(* CoDeSys 2.3.8.0 project: Laser_G67HP_2.pro *)
(* Libraries: STANDARD.LIB 5.6.98 12:03:02 *)

(* Global variable list: Globale_Variablen *)
VAR_GLOBAL

	(* Hardwareeingänge *)
	INot_Aus 			 	AT %IX0.0 : BOOL; (* Eingang 1 *)
	IDruckW			  	AT %IX0.1 : BOOL; (* Eingang 2 *)
	ISchututuer	  		AT %IX0.2 : BOOL; (* Eingang 3 *)
	ISchutzhaube  		AT %IX0.3 : BOOL; (* Eingang 4 *)
	IHWT_EIN			 	AT %IX0.4 : BOOL; (* Eingang 5 *)
	IHWT_AUS			AT %IX0.5 : BOOL; (* Eingang 6 *)
	IHWT_Quitt  			AT %IX0.6 : BOOL; (* Eingang 7 *)
	IRES1					AT %IX0.7 : BOOL; (* Eingang 8 *)

       IINI_Ueberlast  		AT %IX1.0 : BOOL; (* Eingang 9 *)
	IINI_IndexVor	  		AT %IX1.1 : BOOL; (* Eingang 10 *)
	IINI_IndexRueck  		AT %IX1.2 : BOOL; (* Eingang 11 *)
	IINI_Kupplung  		AT %IX1.3 : BOOL; (* Eingang 12 *)
	IRES2			  		AT %IX1.4 : BOOL; (* Eingang 13 *)
	IRES3		 			AT %IX1.5 : BOOL; (* Eingang 14 *)
	IRES4					AT %IX1.6 : BOOL;
	IRES5		 			AT %IX1.7 : BOOL;

	IKammError  			AT %IX2.0 : BOOL; (* Eingang 17 *)
	IKammEnable  		AT %IX2.1 : BOOL; (* Eingang 18 *)
	IKammOutput  		AT %IX2.2 : BOOL; (* Eingang 19 *)
	IRES6		 			AT %IX2.3 : BOOL; (* Eingang 20 *)
	IAbsaug100P 			AT %IX2.4 : BOOL; (* Eingang 21 *)
	IAbsaugFilter			AT %IX2.5 : BOOL; (* Eingang 22 *)
	IRES					AT %IX2.6 : BOOL; (* Eingang 23 *)
	IFU_BB				AT %IX2.7 : BOOL; (* Eingang 24 *)

	IFrgMoma1 			AT %IX3.0 : BOOL;
	IFrgMoma2 			AT %IX3.1 : BOOL;
	IRES7	 				AT %IX3.2 : BOOL;
	IRES8	 				AT %IX3.3 : BOOL;
	ILAS_HWIO 			AT %IX3.4 : BOOL;
	ILAS_SWIO 			AT %IX3.5 : BOOL;
	ILAS_Redy	 		AT %IX3.6 : BOOL;
	ILAS_Res	 			AT %IX3.7 : BOOL;

	ILasDataBit0 			AT %IX4.0 : BOOL;
	ILasDataBit1 	 		AT %IX4.1 : BOOL;
	ILasDataBit2 		 	AT %IX4.2 : BOOL;
	ILasDataBit3 		 	AT %IX4.3 : BOOL;
	ILasDataBit4 	 		AT %IX4.4 : BOOL;
	ILasDataBit5 	 		AT %IX4.5 : BOOL;
	ILasResI1	 		 	AT %IX4.6 : BOOL;
	ILasResI2 			 	AT %IX4.7 : BOOL;

	(*Eingänge für die Panel Tasten*)

	IAPosKS1Input  		AT%IW20:INT;	 	(*Speicher 1 Füllstand analoger Eingang*)
	IARES1				AT%IW22:INT;
	IASSIDgInput			 AT %ID44:UDINT;	(* Drehgeber *)


	QHAmpelGn		 	AT %QX0.0 : BOOL; (* Ventil Pneumatik  *)
	QHAmpelRt	  		AT %QX0.1 : BOOL; (* Ausgang 2 *)
	QHAmpelGb 			AT %QX0.2 : BOOL; (* Ausgang 3 *)
	QRES1				AT %QX0.3 : BOOL; (* Ausgang 4 *)
	QHTasteEin			AT %QX0.4 : BOOL; (* Ausgang 5 *)
	QHTasteAus			AT %QX0.5 : BOOL; (* Ausgang 6 *)
	QHTasteQuitt			AT %QX0.6 : BOOL; (* Ausgang 7 *)
	QRES2				AT %QX0.7 : BOOL; (* Ausgang 8 *)

	QLasMark				AT %QX1.0 : BOOL; (* Ausgang 9 *)
	QLasMarkstop		AT %QX1.1 : BOOL; (* Ausgang 10 *)
	QLasProg1			AT %QX1.2 : BOOL; (* Ausgang 11 *)
	QLasProg2			AT %QX1.3 : BOOL; (* Ausgang 12 *)
	QLasRes2			AT %QX1.4 : BOOL; (* Ausgang 13 *)
	QLasRes3			AT %QX1.5 : BOOL; (* Ausgang 14 *)
	QFrgNaechst			AT %QX1.6 : BOOL; (* Ausgang 15 *)
	QAntriebeEin		     	AT %QX1.7 : BOOL; (* Ausgang 16 *)

	QMotVor	 			AT %QX2.0 : BOOL; (* Ausgang 9 *)
	QMotRueck			AT %QX2.1 : BOOL; (* Ausgang 10 *)
	QSaugAnford			AT %QX2.2 : BOOL; (* Ausgang 11 *)
	QVIndex				AT %QX2.3 : BOOL; (* Ausgang 12 *)
	QVUeberlast			AT %QX2.4 : BOOL; (* Ausgang 13 *)
	QRES5				AT %QX2.5 : BOOL; (* Ausgang 14 *)
	QRES6				AT %QX2.6 : BOOL; (* Ausgang 15 *)
	QRES7			     	AT %QX2.7 : BOOL; (* Ausgang 16 *)

	QASollwMot			AT%QW4:WORD; (*Ausgangswort 1*)
	QARes				 	AT%QW6:WORD; (*Ausgangswort 2*)

(* Anfang der Variablen für Kopmunikation SPS <> Visu *)
	TP_LaserAktiv	:		BOOL;
	TP_LaserHand:			BOOL;
	TP_RefSetzen:			BOOL;
	TP_KammeraAktiv:		BOOL;
	TP_MVor:				BOOL;
	TP_MVorS:				BOOL;
	TP_Mrueck:				BOOL;
	TP_MrueckS:				BOOL;
	TP_Hand:				BOOL;
	TP_Auto:					BOOL;
	TP_ZNullen:				BOOL;   (*not included yet*)
	TPTypIndex:				WORD; (*not included yet*)
	TPTypSpeichern:			BOOL;   (*not included yet*)
	TPKettenTyp: 			ARRAY[0..3] OF WORD;  (*not included yet*)

	S_StUeberlast:			BOOL;
	S_StLaser:				BOOL;
	S_StKammera:			BOOL;
	S_StKupplung	:			BOOL;
	S_StSpeicherSchutz:		BOOL;
	S_StLaserSchutz:			BOOL;
	S_StSpeicher:				BOOL;
	S_StSammelstoerung:	BOOL;
	S_StDruck:				BOOL;
	S_StNotAus:				BOOL;
	S_StRef:					BOOL;

	S_StSchutzTuer:  BOOL;
	S_StSchutzHaube : BOOL;
         S_StAbsaugFilter : BOOL;
         S_StAbsaug100p : BOOL;


	S_MSpeicherVoll:			BOOL;
	S_MSpeicherLeer:		BOOL;
	S_MWarteSpeicher:		BOOL;
	S_MHand:					BOOL;
	S_FKamera:				BOOL;
	S_FLaser:					BOOL;
	S_MAutoStart:				BOOL;
	S_MAutoStop:				BOOL;
	SI_Gliederzahl:			INT;
	SI_ProgNr:				INT;
	SI_IO:						INT;
	SI_NIO:					INT;
	SI_FPosLaser:			INT;
	SI_FPosKamera:			INT;
	SKettenTyp:ARRAY[0..3] OF WORD;  (*not included yet*)
(* ENDE*)

	Skal_IC_SSI_DG_Input: 	DINT;
	Skal_SSI_DG_4:			DINT;
	ZeigerReg:				INT;
	ZeigerKette: 				INT;
	ImpulsPos: 				BOOL;
	ImpulsNeg: 				BOOL;
	Sammelstoerung: BOOL;

	V_Erster_Zyklus: BOOL;
	REF_IO: BOOL;
	AktTypIndexAlt: WORD;
	AktTypindex:WORD;
	PosErreicht: BOOL;


END_VAR

VAR_GLOBAL RETAIN

	(* KettenTyp[0] = Gliederzahl,  Kettentyp[1] Farbe1 0=grau 1=gelb 2=rot 3=blau, Kettentyp[2]=position der ersten Farblasche (Nr.d. Außenlasche*)
	(*Kettentyp[3] Farbe2  Kettentyp[4] Position der zweiten Farblasche *)
	(*Kettentyp[6] Farbe3  Kettentyp[6] Position der dritten Farblasche *)
	(*Kettentyp[7] Farbe4  Kettentyp[8] Position der vierten Farblasche *)
	(*Kettentyp[9] Farbe5  Kettentyp[10] Position der fünften Farblasche *)




	(*Hinterlegte Kettentypen 64 Kettentypen 0-63  , 0=>Gliederzahl, 1-3=>Positionen der ersten bis dritten Außenlasche zum Lasern*)
	(*KettenTyp[x,2]=0 Bedeutet keine zweite Laserung an einer Kette*)
	(*KettenTyp[x,3]=0 Bedeutet keine dritte Laserung an einer Kette*)
	(*KettenTyp[x,1]=0 Nullter Kettentyp keine Laserung*)
	(*KettenTyp[x,0]=0 Ungültiger Eintrag *)

	(*Beispiel für eine Kette: 124 Glieder mit einer Laserung an der ersten Außenlasche gespeichert als Typ 5*)
	(*KettenTyp[5,0]=124   Kettentyp[5,1]=1 Kettentyp[5,2]=0  Kettentyp[5,3]=0*)

	KettenTyp							AT%QW100:ARRAY [0..63,0..3] OF WORD;
	RegMarkierung					AT%QB500:ARRAY[1..500] OF BOOL;


(*   Fehlerzähler für die erste Seite. Fehler können ohne Password zurückgesetzt werden*)

	SI_FKamera				AT%QW70:INT;
	SI_FLaser 				AT%QW72:INT;
(*	ZeigerGlied				AT%QW304:INT;				(* Zeiger für die Glieder in der Anlage zeigt auf das Glied unter der Trennstelle *)
	ZeigerAchtelGlied			AT%QW306:INT;
*)
END_VAR

(* Data type *)
TYPE DriveControl :
STRUCT
	ManOn: BOOL := FALSE; (* Visu -> SPS: Antrieb ein (nur bei FU-Antrieben) *)
	ManOff: BOOL := FALSE; (* Visu -> SPS: Antrieb aus (nur bei FU-Antrieben) *)
	ManFwd: BOOL := FALSE; (* Visu -> SPS: Antrieb im Handbetrieb langsam vorwärts *)
	ManBwd: BOOL := FALSE; (* Visu -> SPS: Antrieb im Handbetrieb langsam rückwärts *)
	TeilungVor: BOOL := FALSE; (* Visu -> SPS: Kette um eine Teilung vor (nur bei Servo-Antrieben) *)
	TeilungZur: BOOL := FALSE; (* Visu -> SPS: Kette um eine Teilung zurück (nur bei Servo-Antrieben) *)
	EnManCtrl: BOOL := FALSE; (* SPS -> Visu: Freigabe manuelle Steuerung *)
	ActOn: BOOL := FALSE; (* SPS -> Visu: Antrieb eingeschaltet *)
	ActOff: BOOL := FALSE; (* SPS -> Visu: Antrieb ausgeschaltet *)
	Error: BOOL := FALSE; (* SPS -> Visu: Störung Antrieb *)
END_STRUCT
END_TYPE

(* Data type *)
TYPE KettenTyp :
STRUCT
	PF: ARRAY [0..19] OF UDINT := 0,410,819,1229,1638,2048,2458,2867,3277,3686,4049,4506,4915,5328,5734,6144,6554,6963,7373,7782;

END_STRUCT
END_TYPE

(* Data type *)
TYPE KS_Control :
STRUCT
	EnInput: BOOL := FALSE; (* Freigabe Befüllen *)
	EnOutput: BOOL := FALSE; (* Freigabe Entleeren *)
	ActState: INT := 0; (* aktueller zustand für Visu *)
END_STRUCT
END_TYPE

(* Data type *)
TYPE KS_Control_1 :
STRUCT
	EnInput: BOOL := FALSE; (* Freigabe Befüllen *)
	EnOutput: BOOL := FALSE; (* Freigabe Entleeren *)
	ActState: INT := 0; (* aktueller zustand für Visu *)
END_STRUCT
END_TYPE

(* Data type *)
TYPE MotorControl :
STRUCT
	ManOn: BOOL := FALSE; (* Visu -> SPS: Antrieb im Handbetrieb ein *)
	ManOff: BOOL := FALSE; (* Visu -> SPS: Antrieb im Handbetrieb aus *)
	EnManCtrl: BOOL := FALSE; (* SPS -> Visu: Freigabe manuelle Steuerung *)
	ActOn: BOOL := FALSE; (* SPS -> Visu: Antrieb eingeschaltet *)
	ActOff: BOOL := FALSE; (* SPS -> Visu: Antrieb ausgeschaltet *)
	Error: BOOL := FALSE; (* SPS -> Visu: Störung Antrieb *)
END_STRUCT
END_TYPE

(* Data type *)
TYPE PneumControl :
STRUCT
	SetOn: BOOL := FALSE; (* Visu -> SPS: Arbeitsstellung anfahren *)
	SetOff: BOOL := FALSE; (* Visu -> SPS: Grundstellung anfahren *)
	EnSet: BOOL := FALSE; (* SPS -> Visu: Freigabe manuell Steuerung *)
	ActOn: BOOL := FALSE; (* SPS -> Visu: Zylinder in Arbeitsstellung *)
	ActOff: BOOL := FALSE; (* SPS -> Visu: Zylinder in Grundstellung *)
	Error: BOOL := FALSE; (* SPS -> Visu: Störung Zylinder oder Endschalter *)
END_STRUCT
END_TYPE

(* Data type *)
TYPE PosControl :
STRUCT
	PosSet: INT := 0; (* Positionssollwert [mm] *)
	ActPos: INT := 0; (* Positionsistwert [mm] *)
	PosLimitLo: INT := 0; (* unterer Grenzwert Sollposition [mm] *)
	PosLimitHi: INT := 0; (* oberer Grenzwert Sollposition [mm] *)
	StartPos: BOOL := FALSE; (* Visu -> SPS: Positionierung starten *)
	StoppPos: BOOL := FALSE; (* Visu -> SPS: Positionierung abbrechen *)
	ManPosUp: BOOL := FALSE; (* Visu -> SPS: Handbetrieb Positon erhöhen *)
	ManPosDn: BOOL := FALSE; (* Visu -> SPS: Handbetrieb Positon verringern *)
	EnPosSet: BOOL := FALSE; (* SPS -> Visu: Freigabe Sollwerteingabe *)
	EnManPos: BOOL := FALSE; (* SPS -> Visu: Freigabe manuelle Positionierung *)
	ActOn: BOOL := FALSE; (* SPS -> Visu: Antrieb eingeschaltet *)
	ActOff: BOOL := FALSE; (* SPS -> Visu: Antrieb ausgeschaltet *)
	Error: BOOL := FALSE; (* SPS -> Visu: Störung Antrieb *)
END_STRUCT
END_TYPE

(* Data type *)
TYPE StationControl :
STRUCT
	StepCounter: INT; (* SPS -> Visu: Schrittzähler *)
	SingleStep: BOOL := FALSE; (* Visu -> SPS: Einzelschritt weiterschalten *)
	SingleCycle: BOOL := FALSE; (* Visu -> SPS: Einzelzyklus ausführen *)
	StartCycle: BOOL := FALSE; (* Zyklus im Auto-Betrieb starten *)
	ManInit: BOOL := FALSE; (* Visu -> SPS: Grundstellung anfahren *)
	AutoInit: BOOL := FALSE; (* Grundstellung im Auto-Betrieb anfahren *)
	SetFinished: BOOL := FALSE; (* Visu -> SPS: Fertigmeldung setzen *)
	WaitPos: BOOL := FALSE; (* Station in Warteposition für Stopp *)
	EnSemiAutoCtrl: BOOL := FALSE; (* SPS -> Visu: Steuerung Halbautomatikbetrieb freigeben; Freigabe für SingleStep, SingleCycle, InitPos und SetFinished *)
	InitPos: BOOL := FALSE; (* Station in Grundstellung *)
	Finished: BOOL := FALSE; (* Station fertig *)
	ErrorInitPos: BOOL := FALSE; (* Störung Grundstellung nicht erreicht *)
	ErrorCycleTime: BOOL := FALSE; (* Störung Zeitüberschreitung Zyklus *)
	ActState: INT := 0; (* SPS -> Visu: Zustand der Station: 0 = Störung, 1 = bereit, 2 = aktiv *)
END_STRUCT
END_TYPE

(* POU INIT, ST *)
PROGRAM INIT

VAR

END_VAR
(* Der Kettentyp wird von Laserrechner ausgewählt *)
AktTypIndex.0:=ILasDataBit0;
AktTypIndex.1:=ILasDataBit1;
AktTypIndex.2:=ILasDataBit2;
AktTypIndex.3:=ILasDataBit3;
AktTypIndex.4:=ILasDataBit4;
AktTypIndex.5:=ILasDataBit5;


(* Wenn Kettentyp gewechselt wurde muß erneut referenziert werden *)
IF AktTypIndex <> AktTypIndexAlt THEN
	REF_IO:=FALSE;
END_IF
AktTypIndexAlt:=AktTypIndex;


(* Wenn die Maschine eingeschaltet wird ist eine Ref Fahrt durchzuführen *)
IF V_Erster_Zyklus=FALSE THEN
	REF_IO:=FALSE;
END_IF
V_Erster_Zyklus:=TRUE;



(* Trennstelle der Kette auf Indexposition fahren und Referenzieren *)
IF REF_IO= FALSE AND TP_RefSetzen= TRUE THEN
	ZeigerKette:=KettenTyp[AktTypIndex,0];
	REF_IO:=TRUE;
END_IF
TP_Refsetzen:=FALSE;
END_PROGRAM

(* POU MAIN_1, FBD *)
PROGRAM MAIN_1
VAR
	SollPos1: SollPos;
	Stufe1: INT;
	ASMSollW1: AsmSollW;
	Poserreicht: BOOL;
	Motorsteuerung1: Motorsteuerun;
	Betriebsarten1: Betriebsarten;
	Kettenspeicher1: Kettenspeicher;
	KSEnIn: BOOL;
	KSEnOut: BOOL;
	Saugersteuerung1: Saugersteuerung;
	Kettentypen1: Kettentypen;
END_VAR
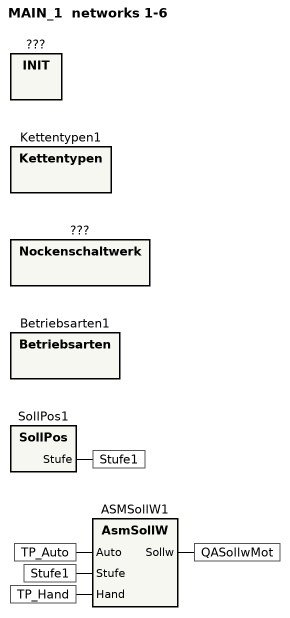
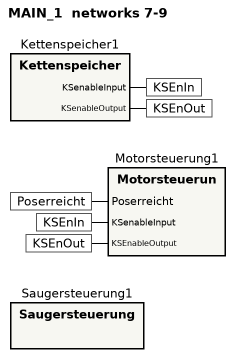
_FBD_ (* Function Block Diagram *)
NETWORK 1
	???:INIT()
NETWORK 2
	Kettentypen1:Kettentypen()
NETWORK 3
	???:Nockenschaltwerk()
NETWORK 4
	Betriebsarten1:Betriebsarten()
NETWORK 5
	SollPos1:SollPos() => Stufe1
NETWORK 6
	ASMSollW1:AsmSollW(Auto: TP_Auto, Stufe: Stufe1, Hand: TP_Hand) => QASollwMot
NETWORK 7
	Kettenspeicher1:Kettenspeicher(KSenableOutput => KSEnOut) => KSEnIn
NETWORK 8
	Motorsteuerung1:Motorsteuerun(Poserreicht: Poserreicht, KSenableInput: KSEnIn, KSEnableOutput: KSEnOut)
NETWORK 9
	Saugersteuerung1:Saugersteuerung()
_END_FBD_
(* the same logic as Structured Text *)
(* Network 1: see the listing above *)
(* Network 2 *)
Kettentypen1();
(* Network 3: see the listing above *)
(* Network 4 *)
Betriebsarten1();
(* Network 5 *)
SollPos1();
Stufe1 := SollPos1.Stufe;
(* Network 6 *)
ASMSollW1(Auto := TP_Auto, Stufe := Stufe1, Hand := TP_Hand);
QASollwMot := ASMSollW1.Sollw;
(* Network 7 *)
Kettenspeicher1();
KSEnOut := Kettenspeicher1.KSenableOutput;
KSEnIn := Kettenspeicher1.KSenableInput;
(* Network 8 *)
Motorsteuerung1(Poserreicht := Poserreicht, KSenableInput := KSEnIn, KSEnableOutput := KSEnOut);
(* Network 9 *)
Saugersteuerung1();
END_PROGRAM

(* POU Funktionsbausteine/SollPos, ST *)
FUNCTION_BLOCK SollPos
VAR_INPUT
END_VAR
VAR_OUTPUT
	Stufe: INT;

END_VAR
VAR
	ZeigerStufe1: INT;
	ZeigerStufe2: INT;
	ZeigerStufe3: INT;
	ZeigerStufe4: INT;
	ZeigerStufe5: INT;
END_VAR
(*
(* Kettenanfang im Handbetrieb setzen *)
IF H_Handbetrieb= TRUE AND TasteKettenanfang=TRUE  THEN
	Zeiger_Kette_Trennstelle:=KettenTyp[0];
	Sperre_2Pruef :=TRUE;
END_IF


(* Auftragswechsel *)

IF	KettenTyp[0] <> Gliederzahl_Alt THEN
	Zeiger_Kette_Trennstelle:= KettenTyp[0];
	Sperre_2Pruef :=TRUE;
END_IF
Gliederzahl_Alt:=KettenTyp[0];
*)


IF	ImpulsPos =TRUE THEN


	(*Alten Eintrag im Register Löschen*)
	(*Laser wird dann die Markierung eintragen*)
	RegMarkierung[ZeigerKette]:=FALSE;

	(* Geschwindigkeitsstufen für die Positionierung ermitteln *)
	(* Zeiger für die Stufen berechnen *)
	(* Bearbeitung nur wenn Aussenlasche*)
	IF ZeigerKette.0=FALSE THEN
		ZeigerStufe1:=ZeigerKette+2;
		IF ZeigerStufe1>KettenTyp[AktTypindex,0] THEN
			ZeigerStufe1:=ZeigerStufe1-KettenTyp[AktTypindex,0];
		END_IF
		ZeigerStufe2:=ZeigerStufe1+2;
		IF ZeigerStufe2>KettenTyp[AktTypindex,0] THEN
			ZeigerStufe2:=ZeigerStufe2-KettenTyp[AktTypindex,0];
		END_IF
		ZeigerStufe3:=ZeigerStufe2+2;
		IF ZeigerStufe3>KettenTyp[AktTypindex,0] THEN
			ZeigerStufe3:=ZeigerStufe3-KettenTyp[AktTypindex,0];
		END_IF
		ZeigerStufe4:=ZeigerStufe3+2;
		IF ZeigerStufe4>KettenTyp[AktTypindex,0] THEN
			ZeigerStufe4:=ZeigerStufe4-KettenTyp[AktTypindex,0];
		END_IF
		ZeigerStufe5:=ZeigerStufe4+2;
		IF ZeigerStufe5>KettenTyp[AktTypindex,0] THEN
			ZeigerStufe5:=ZeigerStufe5-KettenTyp[AktTypindex,0];
		END_IF

		IF ZeigerStufe5 = KettenTyp[AktTypindex,1]*2 OR ZeigerKette = KettenTyp[AktTypindex,2]*2 OR ZeigerKette = KettenTyp[AktTypindex,3]*2THEN
			Stufe:=5;
		ELSE
			Stufe:=6;
		END_IF

		IF ZeigerStufe4 = KettenTyp[AktTypindex,1]*2 OR ZeigerKette = KettenTyp[AktTypindex,2]*2 OR ZeigerKette = KettenTyp[AktTypindex,3]*2THEN
			Stufe:=4;
		END_IF

		IF ZeigerStufe3 = KettenTyp[AktTypindex,1]*2 OR ZeigerKette = KettenTyp[AktTypindex,2]*2 OR ZeigerKette = KettenTyp[AktTypindex,3]*2THEN
			Stufe:=3;
		END_IF

		IF ZeigerStufe2 = KettenTyp[AktTypindex,1]*2 OR ZeigerKette = KettenTyp[AktTypindex,2]*2 OR ZeigerKette = KettenTyp[AktTypindex,3]*2THEN
			Stufe:=2;
		END_IF

		IF ZeigerStufe1 = KettenTyp[AktTypindex,1]*2 OR ZeigerKette = KettenTyp[AktTypindex,2]*2 OR ZeigerKette = KettenTyp[AktTypindex,3]*2THEN
			Stufe:=1;
		END_IF

		IF ZeigerKette = KettenTyp[AktTypindex,1]*2 OR ZeigerKette = KettenTyp[AktTypindex,2]*2 OR ZeigerKette = KettenTyp[AktTypindex,3]*2THEN
		PosErreicht:=TRUE;
		END_IF

	END_IF
END_IF
END_FUNCTION_BLOCK

(* POU Funktionsbausteine/AsmSollW, ST *)
FUNCTION_BLOCK AsmSollW
VAR

END_VAR

VAR_INPUT
	Auto: BOOL;
	Stufe: INT;
	Hand: BOOL;
END_VAR
VAR_OUTPUT
	Sollw: INT;
END_VAR
IF  Auto = TRUE THEN
	Sollw:=Stufe * 5000;
END_IF

IF	Hand=TRUE  THEN
	Sollw:=12000;
END_IF
END_FUNCTION_BLOCK

(* POU Funktionsbausteine/Motorsteuerun, FBD *)
FUNCTION_BLOCK Motorsteuerun
VAR_INPUT
	Poserreicht: BOOL;
	KSenableInput: BOOL;
	KSEnableOutput: BOOL;
END_VAR
VAR_OUTPUT
END_VAR
VAR
	PF_AutoStart: R_TRIG;
	PF_AutoStop: R_TRIG;
	StopGoMot: RS;
END_VAR
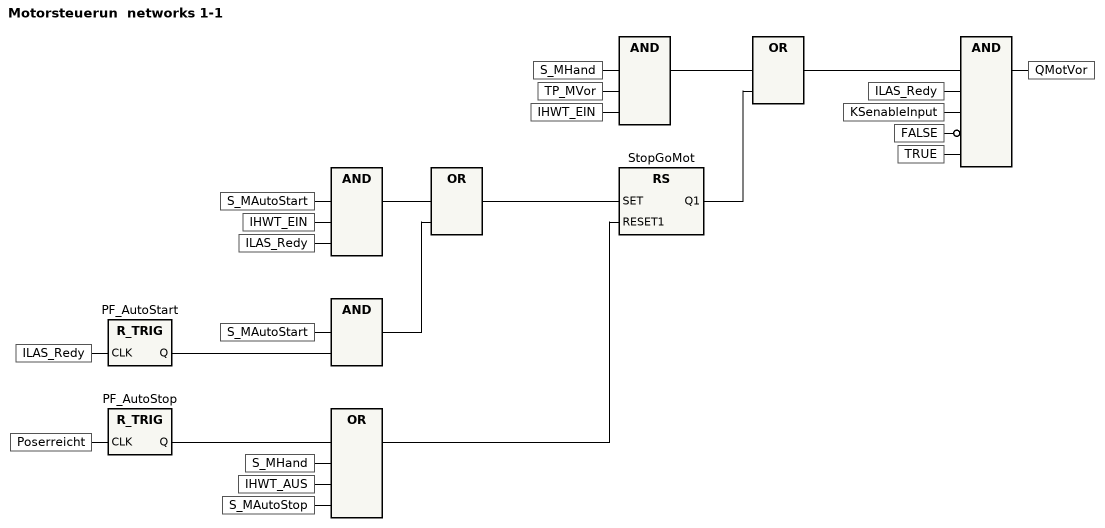
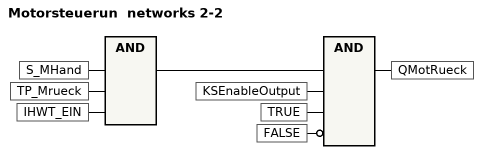
_FBD_ (* Function Block Diagram *)
NETWORK 1 (* Ansteuerung des Motors M1 in Positive richtung *)
	AND(OR(AND(S_MHand, TP_MVor, IHWT_EIN), StopGoMot:RS(SET: OR(AND(S_MAutoStart, IHWT_EIN, ILAS_Redy), AND(S_MAutoStart, PF_AutoStart:R_TRIG(CLK: ILAS_Redy))), RESET1: OR(PF_AutoStop:R_TRIG(CLK: Poserreicht), S_MHand, IHWT_AUS, S_MAutoStop))), ILAS_Redy, KSenableInput, NOT FALSE, TRUE) => QMotVor
NETWORK 2 (* Ansteuerung Motor M1 in negative Richtung *)
	AND(AND(S_MHand, TP_Mrueck, IHWT_EIN), KSEnableOutput, TRUE, NOT FALSE) => QMotRueck
_END_FBD_
(* the same logic as Structured Text *)
(* Network 1: Ansteuerung des Motors M1 in Positive richtung *)
PF_AutoStart(CLK := ILAS_Redy);
PF_AutoStop(CLK := Poserreicht);
StopGoMot(SET := (S_MAutoStart AND IHWT_EIN AND ILAS_Redy) OR (S_MAutoStart AND PF_AutoStart.Q), RESET1 := PF_AutoStop.Q OR S_MHand OR IHWT_AUS OR S_MAutoStop);
QMotVor := ((S_MHand AND TP_MVor AND IHWT_EIN) OR StopGoMot.Q1) AND ILAS_Redy AND KSenableInput AND NOT FALSE AND TRUE;
(* Network 2: Ansteuerung Motor M1 in negative Richtung *)
QMotRueck := (S_MHand AND TP_Mrueck AND IHWT_EIN) AND KSEnableOutput AND TRUE AND NOT FALSE;
END_FUNCTION_BLOCK

(* POU Funktionsbausteine/Betriebsarten, FBD *)
FUNCTION_BLOCK Betriebsarten
VAR_INPUT
END_VAR
VAR_OUTPUT
END_VAR
VAR
END_VAR
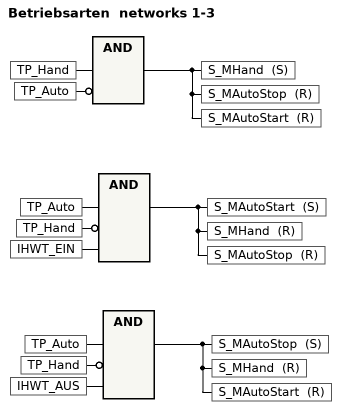
_FBD_ (* Function Block Diagram *)
NETWORK 1
	AND(TP_Hand, NOT TP_Auto) => S S_MHand, R S_MAutoStop, R S_MAutoStart
NETWORK 2
	AND(TP_Auto, NOT TP_Hand, IHWT_EIN) => S S_MAutoStart, R S_MHand, R S_MAutoStop
NETWORK 3
	AND(TP_Auto, NOT TP_Hand, IHWT_AUS) => S S_MAutoStop, R S_MHand, R S_MAutoStart
_END_FBD_
(* the same logic as Structured Text *)
(* Network 1 *)
IF TP_Hand AND NOT TP_Auto THEN S_MHand := TRUE; S_MAutoStop := FALSE; S_MAutoStart := FALSE; END_IF;
(* Network 2 *)
IF TP_Auto AND NOT TP_Hand AND IHWT_EIN THEN S_MAutoStart := TRUE; S_MHand := FALSE; S_MAutoStop := FALSE; END_IF;
(* Network 3 *)
IF TP_Auto AND NOT TP_Hand AND IHWT_AUS THEN S_MAutoStop := TRUE; S_MHand := FALSE; S_MAutoStart := FALSE; END_IF;
END_FUNCTION_BLOCK

(* POU Funktionsbausteine/Kettenspeicher, FBD *)
FUNCTION_BLOCK Kettenspeicher
VAR_INPUT
END_VAR
VAR_OUTPUT
	KSenableInput: BOOL;
	KSenableOutput: BOOL;
END_VAR
VAR
END_VAR
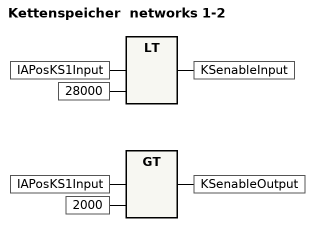
_FBD_ (* Function Block Diagram *)
NETWORK 1
	LT(IAPosKS1Input, 28000) => KSenableInput
NETWORK 2
	GT(IAPosKS1Input, 2000) => KSenableOutput
_END_FBD_
(* the same logic as Structured Text *)
(* Network 1 *)
KSenableInput := IAPosKS1Input < 28000;
(* Network 2 *)
KSenableOutput := IAPosKS1Input > 2000;
END_FUNCTION_BLOCK

(* POU Funktionsbausteine/Saugersteuerung, FBD *)
FUNCTION_BLOCK Saugersteuerung
VAR_INPUT
END_VAR
VAR_OUTPUT
END_VAR
VAR
END_VAR
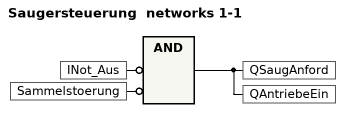
_FBD_ (* Function Block Diagram *)
NETWORK 1
	AND(NOT INot_Aus, NOT Sammelstoerung) => QSaugAnford, QAntriebeEin
_END_FBD_
(* the same logic as Structured Text *)
(* Network 1 *)
QSaugAnford := NOT INot_Aus AND NOT Sammelstoerung;
QAntriebeEin := QSaugAnford;
END_FUNCTION_BLOCK

(* POU Funktionsbausteine/Kettentypen, ST *)
FUNCTION_BLOCK Kettentypen
VAR_INPUT
END_VAR
VAR_OUTPUT
END_VAR
VAR
END_VAR
(*  Angewählten Kettentyp für Visu bereitstellen *)

SKettenTyp[0]:=KettenTyp[TPTypIndex,0];
SKettenTyp[1]:=KettenTyp[TPTypIndex,1];
SKettenTyp[2]:=KettenTyp[TPTypIndex,2];
SKettenTyp[3]:=KettenTyp[TPTypIndex,3];


(* Editierte Kettentypen remanent speichern *)
IF TPTypSpeichern = TRUE THEN
	KettenTyp[TPTypIndex,0]:=TPKettenTyp[0];
	KettenTyp[TPTypIndex,0]:=TPKettenTyp[0];
	KettenTyp[TPTypIndex,0]:=TPKettenTyp[0];
	KettenTyp[TPTypIndex,0]:=TPKettenTyp[0];
END_IF

	TPTypSpeichern:= FALSE;
END_FUNCTION_BLOCK

(* POU Nockenschaltwerk, ST *)
PROGRAM Nockenschaltwerk
VAR
	Zeiger :INT:=0;
	Nocke:BOOL:=FALSE;
	Zaeler:WORD;
	(*Skal_IC_SSI_DG_Input: DINT;*)
	Skal_IC_SSI_DG_Input_Alt:DINT;
	Skal_IC_SSI_DG_Input_Delta:DINT;
	Skal_SSI_DG_4_Alt: DINT;
	ImpulsPos4: BOOL;
END_VAR
(*  Miroslav Knezevic TCM 19.03.07  *)
(* Baustein bildet Zeiger für Speicher (Speichertiefe 500 Glieder) und Zeiger für Kette ( Speichertiefe variabel*)
(* Baustein liefert Impulse bei drehen in positiver Richtung und impulse bei Drehen in negativer Richtung*)
(*  Das Nockenschaltwerk liefert 32 Impulse (32 Glieder(Zähne)  bei einer Umdrehung des SSI Drehgebers *)
(* Voller Kreis = 16777216 Inkremente,  1 Impuls= 524288 Inkremente *)



Skal_IC_SSI_DG_Input:=IASSIDgInput/524288;
Skal_IC_SSI_DG_Input_Delta:=Skal_IC_SSI_DG_Input - Skal_IC_SSI_DG_Input_Alt;


(* Bildung der Virtelgliedimpulse *)
Skal_SSI_DG_4:=IASSIDgInput/131072;
IF Skal_SSI_DG_4 <> Skal_SSI_DG_4_Alt THEN
	ImpulsPos4:=TRUE;
ELSE
	ImpulsPos4:=FALSE;
END_IF
Skal_SSI_DG_4_Alt:=Skal_SSI_DG_4;


IF Skal_IC_SSI_DG_Input_Delta<-10 THEN
	Skal_IC_SSI_DG_Input_Delta:=1;
END_IF

IF Skal_IC_SSI_DG_Input_Delta>10 THEN
	Skal_IC_SSI_DG_Input_Delta:=-1;
END_IF


ZeigerReg:=DINT_TO_INT(ZeigerReg+Skal_IC_SSI_DG_Input_Delta);
IF ZeigerReg>500 THEN
	ZeigerReg:=ZeigerReg-500;
END_IF
IF ZeigerReg<1 THEN
	ZeigerReg:=ZeigerReg+500;
END_IF


ZeigerKette:=DINT_TO_INT(ZeigerKette+Skal_IC_SSI_DG_Input_Delta);
IF ZeigerKette>KettenTyp[AktTypindex,0] THEN
	ZeigerKette:=ZeigerKette-KettenTyp[AktTypindex,0];
END_IF

IF ZeigerKette<1 THEN
	ZeigerKette:=ZeigerKette-KettenTyp[AktTypindex,0];
END_IF


IF Skal_IC_SSI_DG_Input_Delta>0 THEN
	ImpulsPos:=TRUE;
ELSE
	ImpulsPos:=FALSE;
END_IF;

IF Skal_IC_SSI_DG_Input_Delta<0 THEN
	ImpulsNeg:=TRUE;
ELSE
	ImpulsNeg:=FALSE;
END_IF;



Skal_IC_SSI_DG_Input_Alt:=Skal_IC_SSI_DG_Input;
END_PROGRAM

(* POU MAIN_2, ST *)
PROGRAM MAIN_2
VAR
END_VAR
;
END_PROGRAM

(* POU Funktionsbausteine/Indexsteuernung, FBD *)
FUNCTION_BLOCK Indexsteuernung
VAR_INPUT
END_VAR
VAR_OUTPUT
END_VAR
VAR
	SR1: RS;
	PF_1: R_TRIG;
	PF2: R_TRIG;
	PF_3: R_TRIG;
END_VAR
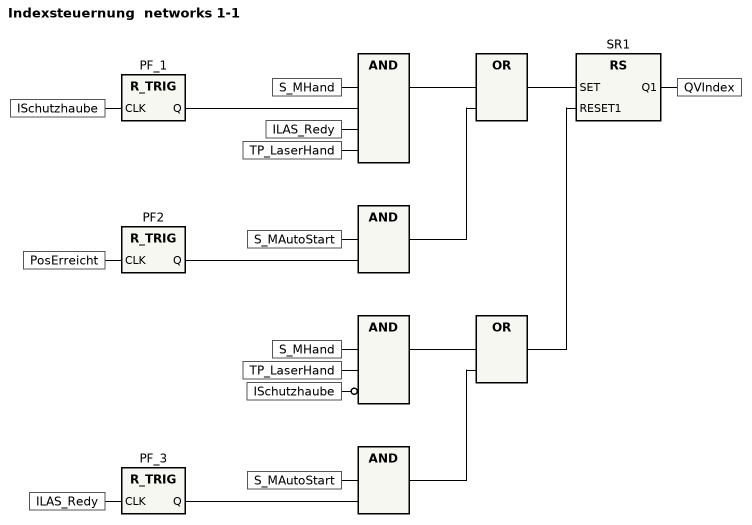
_FBD_ (* Function Block Diagram *)
NETWORK 1
	SR1:RS(SET: OR(AND(S_MHand, PF_1:R_TRIG(CLK: ISchutzhaube), ILAS_Redy, TP_LaserHand), AND(S_MAutoStart, PF2:R_TRIG(CLK: PosErreicht))), RESET1: OR(AND(S_MHand, TP_LaserHand, NOT ISchutzhaube), AND(S_MAutoStart, PF_3:R_TRIG(CLK: ILAS_Redy)))) => QVIndex
_END_FBD_
(* the same logic as Structured Text *)
(* Network 1 *)
PF_1(CLK := ISchutzhaube);
PF2(CLK := PosErreicht);
PF_3(CLK := ILAS_Redy);
SR1(SET := (S_MHand AND PF_1.Q AND ILAS_Redy AND TP_LaserHand) OR (S_MAutoStart AND PF2.Q), RESET1 := (S_MHand AND TP_LaserHand AND NOT ISchutzhaube) OR (S_MAutoStart AND PF_3.Q));
QVIndex := SR1.Q1;
END_FUNCTION_BLOCK
